TYPE ST_DeviceState :
STRUCT
	bDeviceCommOK		: BOOL;
	bDeviceEnabled		: BOOL;
	bDeviceEnableCmd	: BOOL;
	bDeviceFaulted		: BOOL;
	bDeviceReset		: BOOL;
	nDeviceStatusFeedback	: DWORD; // Mapped from the hardware status registry. Size depends on the config
END_STRUCT
END_TYPE

(* stored: Version 1.1.0.1
   DUT ST_DeviceState: Id {e6bb178d-59b1-4bd4-95a8-c8ce46e5aa65} *)
